// TwinCAT 3 PLC project Main
// ProgramVersion: 3.1.4023.0
// libraries:
//   Tc2_MC2, * (Beckhoff Automation GmbH)
//   Tc2_Standard, * (Beckhoff Automation GmbH)
//   Tc2_System, * (Beckhoff Automation GmbH)
//   Tc3_Module, * (Beckhoff Automation GmbH)
//   VisuDialogs, * (System)
//   VisuSymbols,3.5.10.0,System
// project tree:
//   DUTs/Control/ ForceControlParam.TcDUT, JogParam.TcDUT
//   DUTs/Converter/ MotorDegreeToCablePositionParam.TcDUT
//   DUTs/ MotorParam.TcDUT, MotorState.TcDUT, SensorData.TcDUT, SystemControlMode.TcDUT, SystemControlParam.TcDUT
//   / GlobalTextList.TcGTLO, PlcTask.TcTTO, 视图管理器.TcVMO (not stored)
//   GVLs/ GVL.TcGVL
//   POUs/Converter/ MotorDegreeToCablePosition.TcPOU, CableVelocityToMotorAngularVelocity.TcPOU, MotorAngularVelocityToCableVelocity.TcPOU
//   POUs/ MAIN.TcPOU, SystemControl.TcPOU
//   POUs/Safety/ VelocitySaturation.TcPOU
//   VISUs/ ControlHMI.TcVIS
// real-time tasks:
//   TASK PlcTask: cycle T#1ms, priority 20, ADS port 350
// motion (NC):
//   TASK NC-Task 1 SAF: cycle T#1ms, priority 4, ADS port 501
//   TASK NC-Task 1 SVB: cycle T#1ms, priority 8, ADS port 511
//   AXIS Axis 1 (id 1)
//     General: UnitName=Degree
//     Dynamic: AccelerationMaximum=540, DecelerationMaximum=540, Acceleration=540, Deceleration=540, Jerk=1620
//     Velo: RefSearch=180, RefSync=180, SlowManual=60, FastManual=120, Fast=18075.9448242188, Maximum=360
//     PositionAreaControl: Enable=false
//     TargetPosControl: Enable=false
//     OtherSettings: AllowMotionCmdToSlave=true
//     encoder EncType=8
//       EncPara: ScaleFactorNumerator=360, ScaleFactorDenominator=1048576, MaxCount=#xffffffff
//     drive DrvType=9
//       DrvPara: MaxCount=#xffffffff, DriveControlDWord=#x00030000
//         Analog: VeloReferenz=360, VeloScale=1.02400649589962, TorqueSetpointScale=10, ScaleFactorActTorque=0.1
//         TimeComp: TaskDelayCycles=1
//     controller CtrType=1
//       CtrPara: PriorControlFactor=1
//         PosDiffControl: Enable=false
//         Observer: BandWidth=20
// I/O:
//   DEVICE Device 3 (EtherCAT), AmsNetId 192.168.137.1.4.1
//     Term 1 (EK1100) [EK1100 EtherCAT Coupler (2A E-Bus)]
//       Term 2 (EL9505) [EL9505 Power supply terminal 5V]
//       Term 3 (EL3356) [EL3356 1Ch. Ana. Input Resistor Bridge Terminal, 16bit, High Precision]
//       Term 5 (EL9011) [EL9011 End Terminal]
//     Drive 4 (AX5106-0000-0203) [AX5106-0000-0203 EtherCAT Drive (SoE, 1 Ch.)]
// variable links:
//   Main/Main Instance <-> Device 3 (EtherCAT)/Drive 4 (AX5106-0000-0203)
//     PlcTask Outputs/MAIN.motor_param.target_axis_velocity_raw <-> MDT/Velocity command value
//   Main/Main Instance <-> Device 3 (EtherCAT)/Term 1 (EK1100)/Term 3 (EL3356)
//     PlcTask Inputs/MAIN.sensor_data.force_value_raw <-> RMB Value (Real)/Value (Real)
//   Main/Main Instance <-> NC-Task 1 SAF/Axes/Axis 1
//     PlcTask Inputs/GVL.axis1.NcToPlc <-> Outputs/ToPlc
//     PlcTask Outputs/GVL.axis1.PlcToNc <-> Inputs/FromPlc
//   (this object) <-> Device 3 (EtherCAT)/Drive 4 (AX5106-0000-0203)
//     Drive/Inputs/In/nDataIn3[0] <-> AT/Torque feedback value
//     Drive/Inputs/In/nDcOutputTime <-> InfoData/DcOutputShift
//     Drive/Inputs/In/nState1 <-> AT/Drive status word @bit 8
//     Drive/Inputs/In/nState2 <-> AT/Drive status word
//     Drive/Inputs/In/nState4 @bit 1 <-> WcState/InputToggle
//     Drive/Inputs/In/nState4 <-> WcState/WcState
//     Drive/Outputs/Out/nCtrl1 <-> MDT/Master control word @bit 8
//     Enc/Inputs/In/nDataIn1 <-> AT/Position feedback value 1 (motor feedback)
//     Enc/Inputs/In/nDataIn7 <-> AT/Velocity feedback value 1
//     Enc/Inputs/In/nDcInputTime <-> InfoData/DcInputShift
//     Enc/Inputs/In/nState4 @bit 1 <-> WcState/InputToggle
//     Enc/Inputs/In/nState4 <-> WcState/WcState

CONFIGURATION Main
    RESOURCE PLC ON TwinCAT3
        TASK PlcTask(INTERVAL := T#1ms, PRIORITY := 20);
        PROGRAM MAIN WITH PlcTask : MAIN;
    END_RESOURCE
END_CONFIGURATION

// ---- DUTs/Control/ForceControlParam.TcDUT
TYPE ForceControlParam :
STRUCT

END_STRUCT
END_TYPE

// ---- DUTs/Control/JogParam.TcDUT
TYPE JogParam :
STRUCT
	jog_velocity : LREAL;
END_STRUCT
END_TYPE

// ---- DUTs/Converter/MotorDegreeToCablePositionParam.TcDUT
TYPE MotorDegreeToCablePositionParam :
STRUCT
	reset_cable_position : BOOL;
END_STRUCT
END_TYPE

// ---- DUTs/MotorParam.TcDUT
TYPE MotorParam :
STRUCT
	// 发送给电机的速度
	target_axis_velocity_raw AT %Q* : DINT;
	
	// 期望的放绳速度
	target_cable_velocity : LREAL;
	
	// 最大最小速度(mm/s)
	max_cable_velocity : LREAL := 200;
	min_cable_velocity : LREAL := -200;
END_STRUCT
END_TYPE

// ---- DUTs/MotorState.TcDUT
TYPE MotorState :
STRUCT
	// 原始电机位置、速度，直接从axis返回
	axis_position_raw : LREAL;
	axis_velocity_raw : LREAL;
	
	// 电机位置、速度，转换为放绳量，单位mm
	cable_position : LREAL;
	cable_velocity : LREAL;
	
	// 电机驱动器状态
	is_motor_closedloop : BOOL;		// 电机是否已经进入闭环使能状态，可以进行运动控制
END_STRUCT
END_TYPE

// ---- DUTs/SensorData.TcDUT
TYPE SensorData :
STRUCT
	force_value_raw AT %I* : REAL;
END_STRUCT
END_TYPE

// ---- DUTs/SystemControlMode.TcDUT
{attribute 'qualified_only'}
{attribute 'strict'}
TYPE SystemControlMode :
(
	Debug := 0,
	ConstForce := 1
);
END_TYPE

// ---- DUTs/SystemControlParam.TcDUT
TYPE SystemControlParam :
STRUCT
	is_motor_poweron : BOOL;
	is_system_exit : BOOL;
	is_system_control : BOOL;
	system_control_mode : SystemControlMode;
	
	// Debug
	is_motor_jog : BOOL;
	jog_param : JogParam;
	// ConstForce
	is_force_control : BOOL;
	force_control_param : ForceControlParam;
	
	// Other Param
	motor_degree2cable_position_param : MotorDegreeToCablePositionParam;
END_STRUCT
END_TYPE

// ---- GVLs/GVL.TcGVL
{attribute 'qualified_only'}
VAR_GLOBAL
	axis1 : Tc2_MC2.AXIS_REF;
END_VAR

// ---- POUs/MAIN.TcPOU
PROGRAM MAIN
VAR
	sensor_data : SensorData;
	MotorDegreeToCablePosition : MotorDegreeToCablePosition;	

	SystemControl : SystemControl;
	system_control_param : SystemControlParam;
	motor_state : MotorState;
	motor_param : MotorParam;
END_VAR

// 系统状态读取
GVL.axis1.ReadStatus();
motor_state.is_motor_closedloop := GVL.axis1.Status.ControlLoopClosed;
motor_state.axis_position_raw := GVL.axis1.NcToPlc.ActPos;
motor_state.axis_velocity_raw := GVL.axis1.NcToPlc.ActVelo;

// 电机参数转换
MotorDegreeToCablePosition(
	motor_position:= motor_state.axis_position_raw, 
	reset_cable_position:= system_control_param.motor_degree2cable_position_param.reset_cable_position, 
	cable_position=> motor_state.cable_position);
MotorAngularVelocityToCableVelocity(motor_velocity:= motor_state.axis_velocity_raw, cable_velocity=> motor_state.cable_velocity);

// 控制状态机
SystemControl(
	motor_axis:= GVL.axis1, 
	system_control_param:= system_control_param, 
	motor_state:= motor_state, 
	target_velocity=> motor_param.target_cable_velocity);

// 安全限制 
VelocitySaturation(
	velocity:= motor_param.target_cable_velocity, 
	max_velocity:= motor_param.max_cable_velocity, 
	min_velocity:= motor_param.min_cable_velocity);

// 电机参数转换
CableVelocityToMotorAngularVelocity(cable_velocity:= motor_param.target_cable_velocity, motor_velocity=> motor_param.target_axis_velocity_raw);

END_PROGRAM

// ---- POUs/Converter/MotorDegreeToCablePosition.TcPOU
FUNCTION_BLOCK MotorDegreeToCablePosition
VAR_IN_OUT
	motor_position : LREAL;	// deg/s
	reset_cable_position : BOOL;	
END_VAR
VAR_OUTPUT
	cable_position : LREAL;
END_VAR
VAR
	winch_radius : LREAL := 16.0;
END_VAR
VAR PERSISTENT
	motor_position_shift : LREAL;
END_VAR

IF reset_cable_position THEN
	motor_position_shift := motor_position;
END_IF

cable_position := (motor_position - motor_position_shift) * Tc2_System.PI / 180.0 * winch_radius;

END_FUNCTION_BLOCK

// ---- POUs/SystemControl.TcPOU
FUNCTION_BLOCK SystemControl
VAR_IN_OUT
	motor_axis : Tc2_MC2.AXIS_REF;
	system_control_param : SystemControlParam;
	motor_state : MotorState;
END_VAR
VAR_OUTPUT
	target_velocity : LREAL;
END_VAR
VAR
	motorPower : Tc2_MC2.MC_Power;
END_VAR

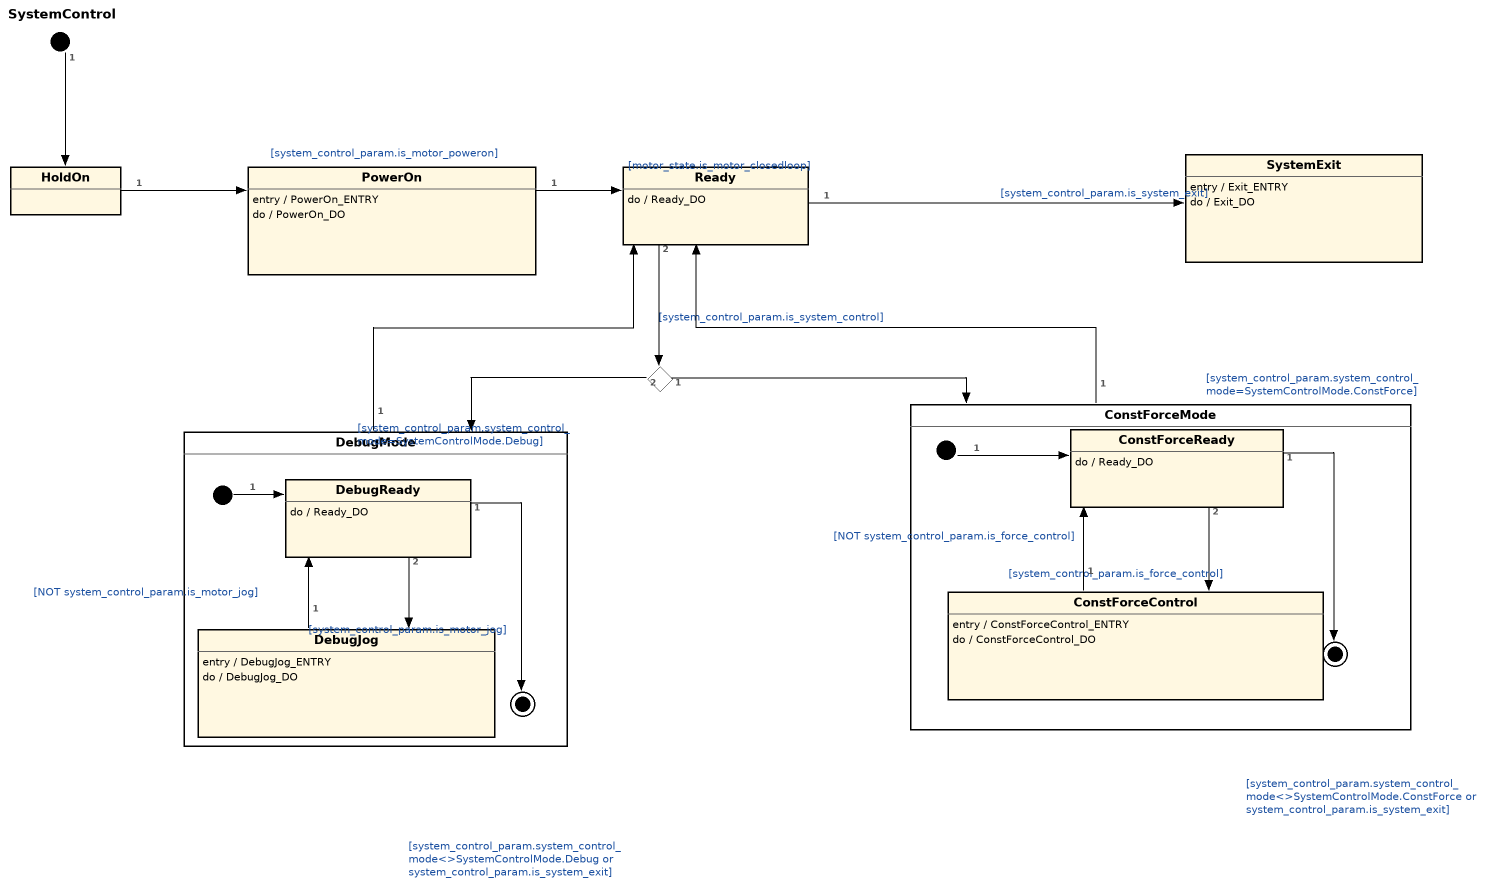
STATECHART SystemControl  // abortable
    START StartState1
    STATE HoldOn
    STATE PowerOn
        entry / PowerOn_ENTRY
        do / PowerOn_DO
    STATE Ready
        do / Ready_DO
    STATE SystemExit
        entry / Exit_ENTRY
        do / Exit_DO
    CHOICE ChoiceElement1
    COMPOSITE STATE ConstForceMode
        START StartState3
        STATE ConstForceReady
            do / Ready_DO
        STATE ConstForceControl
            entry / ConstForceControl_ENTRY
            do / ConstForceControl_DO
        END EndState2
        StartState3 -> ConstForceReady  // priority 1, on completion
        ConstForceReady -> EndState2 [system_control_param.system_control_mode<>SystemControlMode.ConstForce or system_control_param.is_system_exit] // priority 1
        ConstForceReady -> ConstForceControl [system_control_param.is_force_control] // priority 2
        ConstForceControl -> ConstForceReady [NOT system_control_param.is_force_control] // priority 1
    END_STATE
    COMPOSITE STATE DebugMode
        START StartState2
        STATE DebugReady
            do / Ready_DO
        STATE DebugJog
            entry / DebugJog_ENTRY
            do / DebugJog_DO
        END EndState1
        StartState2 -> DebugReady  // priority 1, on completion
        DebugReady -> EndState1 [system_control_param.system_control_mode<>SystemControlMode.Debug or system_control_param.is_system_exit] // priority 1
        DebugReady -> DebugJog [system_control_param.is_motor_jog] // priority 2
        DebugJog -> DebugReady [NOT system_control_param.is_motor_jog] // priority 1
    END_STATE
    StartState1 -> HoldOn  // priority 1, on completion
    HoldOn -> PowerOn [system_control_param.is_motor_poweron] // priority 1
    PowerOn -> Ready [motor_state.is_motor_closedloop] // priority 1
    Ready -> SystemExit [system_control_param.is_system_exit] // priority 1
    Ready -> ChoiceElement1 [system_control_param.is_system_control] // priority 2
    ChoiceElement1 -> ConstForceMode [system_control_param.system_control_mode=SystemControlMode.ConstForce] // priority 1
    ChoiceElement1 -> DebugMode [system_control_param.system_control_mode=SystemControlMode.Debug] // priority 2
    ConstForceMode -> Ready  // priority 1, on completion
    DebugMode -> Ready  // priority 1, on completion
END_STATECHART

ACTION ConstForceControl_DO:

END_ACTION

ACTION ConstForceControl_ENTRY:

END_ACTION

ACTION DebugJog_DO:
target_velocity := system_control_param.jog_param.jog_velocity;
END_ACTION

ACTION DebugJog_ENTRY:

END_ACTION

ACTION Exit_DO:
motorPower(
	Axis:= motor_axis, 
	Enable:= FALSE, 
	Enable_Positive:= TRUE, 
	Enable_Negative:= TRUE, 
	Override:= , 
	BufferMode:= , 
	Options:= , 
	Status=> , 
	Busy=> , 
	Active=> , 
	Error=> , 
	ErrorID=> );
END_ACTION

ACTION Exit_ENTRY:
target_velocity := 0;
END_ACTION

ACTION PowerOn_DO:
motorPower(
	Axis:= motor_axis, 
	Enable:= TRUE, 
	Enable_Positive:= TRUE, 
	Enable_Negative:= TRUE, 
	Override:= , 
	BufferMode:= , 
	Options:= , 
	Status=> , 
	Busy=> , 
	Active=> , 
	Error=> , 
	ErrorID=> );
END_ACTION

ACTION PowerOn_ENTRY:

END_ACTION

ACTION Ready_DO:
target_velocity := 0;
END_ACTION

END_FUNCTION_BLOCK

// ---- POUs/Converter/MotorAngularVelocityToCableVelocity.TcPOU
FUNCTION MotorAngularVelocityToCableVelocity : LREAL
VAR_INPUT
	motor_velocity : LREAL;	// deg/s
END_VAR
VAR_OUTPUT
	cable_velocity : LREAL;
END_VAR
VAR
	winch_radius : LREAL := 16.0;
END_VAR

cable_velocity := motor_velocity * Tc2_System.PI / 180.0 * winch_radius;

END_FUNCTION

// ---- POUs/Safety/VelocitySaturation.TcPOU
FUNCTION VelocitySaturation : LREAL
VAR_IN_OUT
	velocity : LREAL;
	max_velocity : LREAL;
	min_velocity : LREAL;
END_VAR

IF velocity > max_velocity THEN
	velocity := max_velocity;
END_IF
IF velocity < min_velocity THEN
	velocity := min_velocity;
END_IF

END_FUNCTION

// ---- POUs/Converter/CableVelocityToMotorAngularVelocity.TcPOU
FUNCTION CableVelocityToMotorAngularVelocity : LREAL
VAR_INPUT
	cable_velocity : LREAL;
END_VAR
VAR_OUTPUT
	motor_velocity : DINT;
END_VAR
VAR
	velocity_ratio : LREAL := 17895.697;	// motor unit: rev/(2^30 ms) => 1 rpm = 17895.697 unit
	winch_radius : LREAL := 16.0;
END_VAR

// calculation: cable_velocity/winch_radius/pi*180*60/360 rpm 
motor_velocity := LREAL_TO_DINT(cable_velocity / winch_radius * 30.0 /Tc2_System.PI * velocity_ratio);

END_FUNCTION

// ---- GlobalTextList.TcGTLO
TEXTLIST GlobalTextList
  450 = '%5.2f'
  855 = 'ConstForce'
  81 = 'Debug'
  497 = 'Debug 模式配置'
  258 = 'Debug模式'
  259 = 'Force 模式配置'
  177 = 'Force模式'
  202 = '使能电机'
  681 = '力传感器信号'
  119 = '反向最大速度'
  322 = '开始控制'
  142 = '控制模式选择'
  6 = '正向最大速度'
  217 = '点动电机'
  797 = '点动速度'
  717 = '电机位置'
  856 = '电机使能'
  933 = '电机速度'
  94 = '系统配置'
  212 = '系统默认配置'
  5 = '绳索速度'
  875 = '绳索长度'
  74 = '退出系统'
  988 = '重置绳长'
END_TEXTLIST

// ---- VISUs/ControlHMI.TcVIS
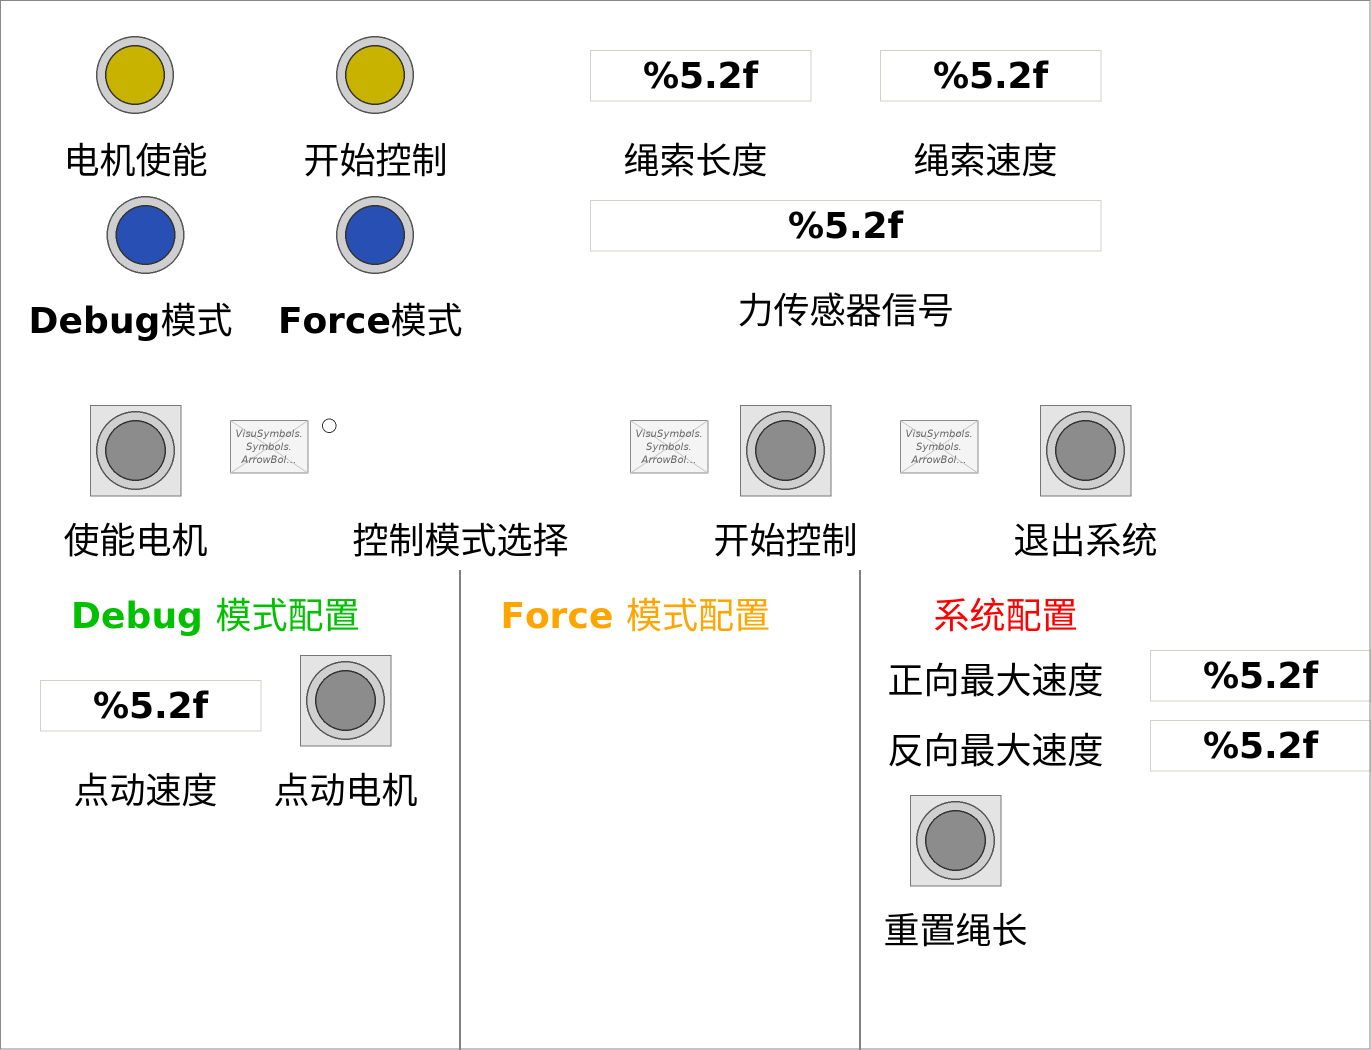
VISUALIZATION ControlHMI  // 1371x1050
    Lamp1 (90,30 90x90), variable: Main.motor_state.is_motor_closedloop, style: Lamp-Lamp1-Yellow
    Label (40,130 191x61), "电机使能"
    Lamp1 (330,30 90x90), variable: Main.system_control_param.is_system_control, style: Lamp-Lamp1-Yellow
    Label (280,130 191x61), "开始控制"
    Label (20,290 221x61), "Debug模式"
    Lamp1 (100,190 91x90), variable: Main.system_control_param.system_control_mode=SystemControlMode.Debug, style: Lamp-Lamp1-Blue
    Label (260,290 221x61), "Force模式"
    Lamp1 (330,190 90x90), variable: Main.system_control_param.system_control_mode=SystemControlMode.ConstForce, style: Lamp-Lamp1-Blue
    Textfield (590,50 221x51), "%5.2f", text variable: Main.motor_state.cable_position
    Label (600,130 191x61), "绳索长度"
    Label (890,130 191x61), "绳索速度"
    Textfield (880,50 221x51), "%5.2f", text variable: Main.motor_state.cable_velocity
    Label (600,280 491x61), "力传感器信号"
    Textfield (590,200 511x51), "%5.2f", text variable: Main.sensor_data.force_value_raw
    PushSwitchLed (90,400 91x101), variable: Main.system_control_param.is_motor_poweron, behaviour: TAP, style: Switch-PushSwitchLed-Gray
    Label (40,510 191x61), "使能电机"
    Image (230,420 78x53), image: VisuSymbols.Symbols.ArrowBoldRight
    RadioButton (320,340 301x171), variable: Main.system_control_param.system_control_mode
        Areas[0]: Text=Debug
        Areas[1]: Text=ConstForce
    Label (310,510 301x61), "控制模式选择"
    Image (630,420 78x53), image: VisuSymbols.Symbols.ArrowBoldRight
    PushSwitchLed (740,400 91x101), variable: Main.system_control_param.is_system_control, behaviour: TOGGLE, style: Switch-PushSwitchLed-Gray
    Label (690,510 191x61), "开始控制"
    Line (460,1050) (460,570)
    PushSwitchLed (1040,400 91x101), variable: Main.system_control_param.is_system_exit, behaviour: TOGGLE, style: Switch-PushSwitchLed-Gray
    Label (990,510 191x61), "退出系统"
    Image (900,420 78x53), image: VisuSymbols.Symbols.ArrowBoldRight
    Label (40,580 351x71), "Debug 模式配置"
    Label (250,760 191x61), "点动电机"
    PushSwitchLed (300,650 91x101), variable: Main.system_control_param.is_motor_jog, behaviour: TAP, style: Switch-PushSwitchLed-Gray
    Textfield (40,680 221x51), "%5.2f", text variable: Main.system_control_param.jog_param.jog_velocity
        OnMouseClick: write the text variable via Default
    Label (50,760 191x61), "点动速度"
    Label (460,580 351x71), "Force 模式配置"
    Line (860,1050) (860,570)
    Label (830,580 351x71), "系统配置"
    Textfield (1150,650 221x51), "%5.2f", text variable: Main.motor_param.max_cable_velocity
        OnMouseClick: write the text variable via Default
    Label (860,650 271x61), "正向最大速度"
    Label (860,720 271x61), "反向最大速度"
    Textfield (1150,720 221x51), "%5.2f", text variable: Main.motor_param.min_cable_velocity
        OnMouseClick: write the text variable via Default
    PushSwitchLed (910,790 91x101), variable: Main.system_control_param.motor_degree2cable_position_param.reset_cable_position, behaviour: TAP, style: Switch-PushSwitchLed-Gray
    Label (860,900 191x61), "重置绳长"
END_VISUALIZATION
